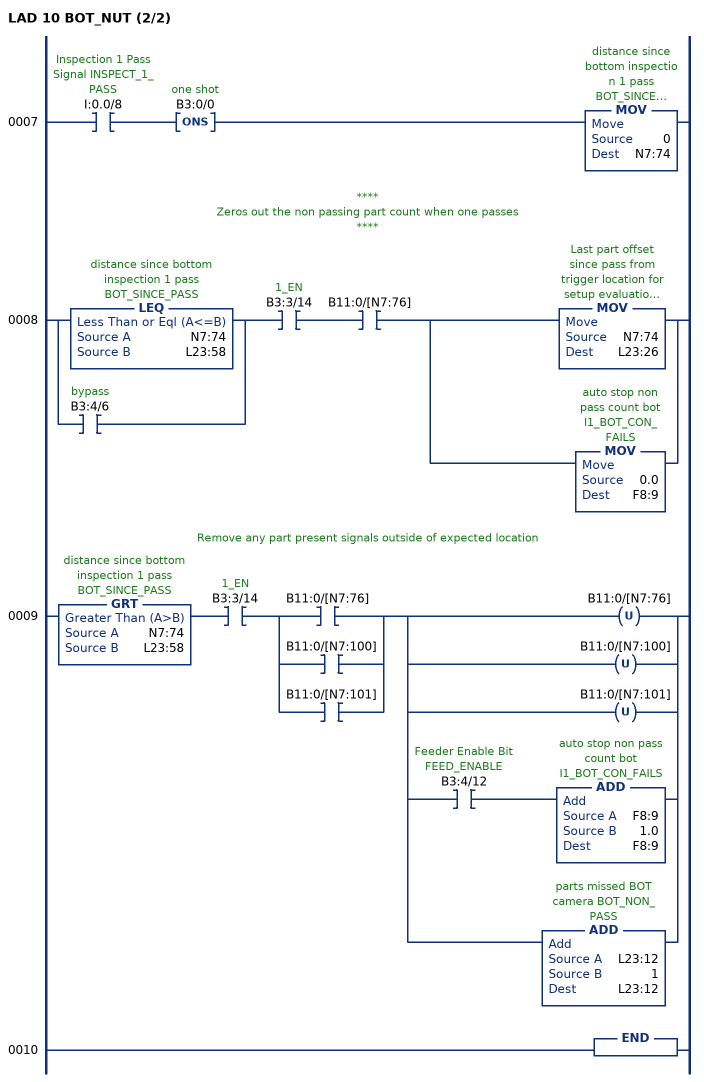
% Rung: 7 %
SOR XIC I:0.0/8 ONS B3:0/0 MOV 0 N7:74 EOR
%   I:0.0/8  INSPECT_1_PASS  "Inspection 1 Pass Signal" %
%   B3:0/0  "one shot" %
%   N7:74  BOT_SINCE_PASS  "distance since bottom inspection 1 pass" %
% Rung: 8 %
% ****
%                   Zeros out the non passing part count when one passes
% **** %
SOR BST LEQ N7:74 L23:58 NXB XIC B3:4/6 BND XIC B3:3/14 XIC B11:0/[N7:76] BST MOV N7:74 L23:26 NXB MOV 0.0 F8:9 BND EOR
%   N7:74  BOT_SINCE_PASS  "distance since bottom inspection 1 pass" %
%   L23:58  BOT_RES_WIDTH %
%   B3:4/6  "bypass" %
%   B3:3/14  1_EN %
%   N7:76  BOT_TEST_LOC  "Location of pass window." %
%   L23:26  LAST_BOT_OFFSET  "Last part offset since pass from trigger location for setup evaluation" %
%   F8:9  I1_BOT_CON_FAILS  "auto stop non pass count bot" %
% Rung: 9 %
% Remove any part present signals outside of expected location %
SOR GRT N7:74 L23:58 XIC B3:3/14 BST XIC B11:0/[N7:76] NXB XIC B11:0/[N7:100] NXB XIC B11:0/[N7:101] BND BST BST OTU B11:0/[N7:76] NXB OTU B11:0/[N7:100] NXB OTU B11:0/[N7:101] BND NXB XIC B3:4/12 ADD F8:9 1.0 F8:9 NXB ADD L23:12 1 L23:12 BND EOR
%   N7:74  BOT_SINCE_PASS  "distance since bottom inspection 1 pass" %
%   L23:58  BOT_RES_WIDTH %
%   B3:3/14  1_EN %
%   N7:76  BOT_TEST_LOC  "Location of pass window." %
%   B3:4/12  FEED_ENABLE  "Feeder Enable Bit" %
%   F8:9  I1_BOT_CON_FAILS  "auto stop non pass count bot" %
%   L23:12  BOT_NON_PASS  "parts missed BOT camera" %
% Rung: 10 %
SOR END EOR

LADDER 11 "DATA_TRANS"
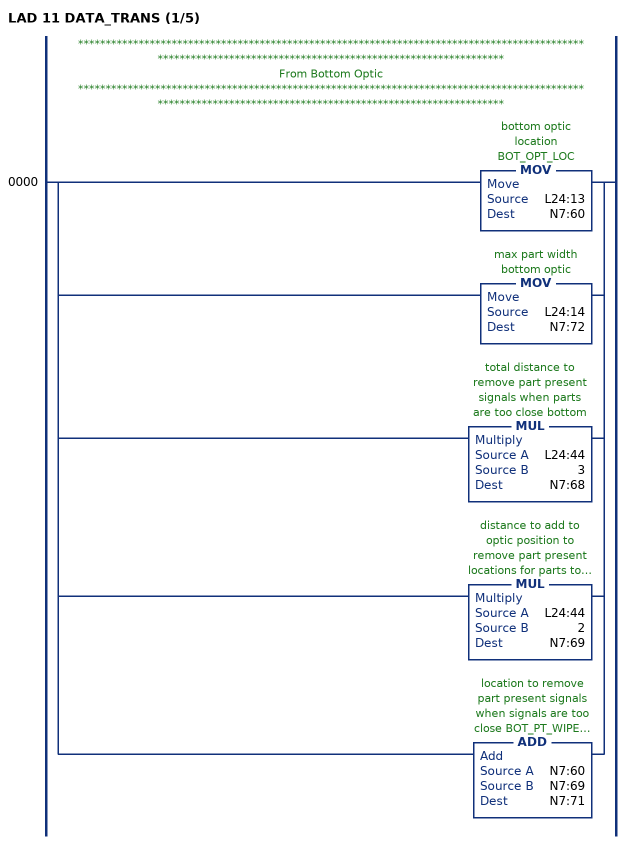
% Rung: 0 %
% ***********************************************************************************************************************************************************
% From Bottom Optic
% *********************************************************************************************************************************************************** %
SOR BST BST MOV L24:13 N7:60 NXB MOV L24:14 N7:72 BND NXB MUL L24:44 3 N7:68 NXB MUL L24:44 2 N7:69 NXB ADD N7:60 N7:69 N7:71 BND EOR
%   L24:13  BOT_OPTIC_LOC %
%   N7:60  BOT_OPT_LOC  "bottom optic location" %
%   L24:14  MAX_PART_WIDTH_BOT %
%   N7:72  "max part width bottom optic" %
%   L24:44  MIN_PART_GAP_BOT %
%   N7:68  "total distance to remove part present signals when parts are too close bottom" %
%   N7:69  "distance to add to optic position to remove part present locations for parts too close bottom" %
%   N7:71  BOT_PT_WIPE_LOC  "location to remove part present signals when signals are too close" %

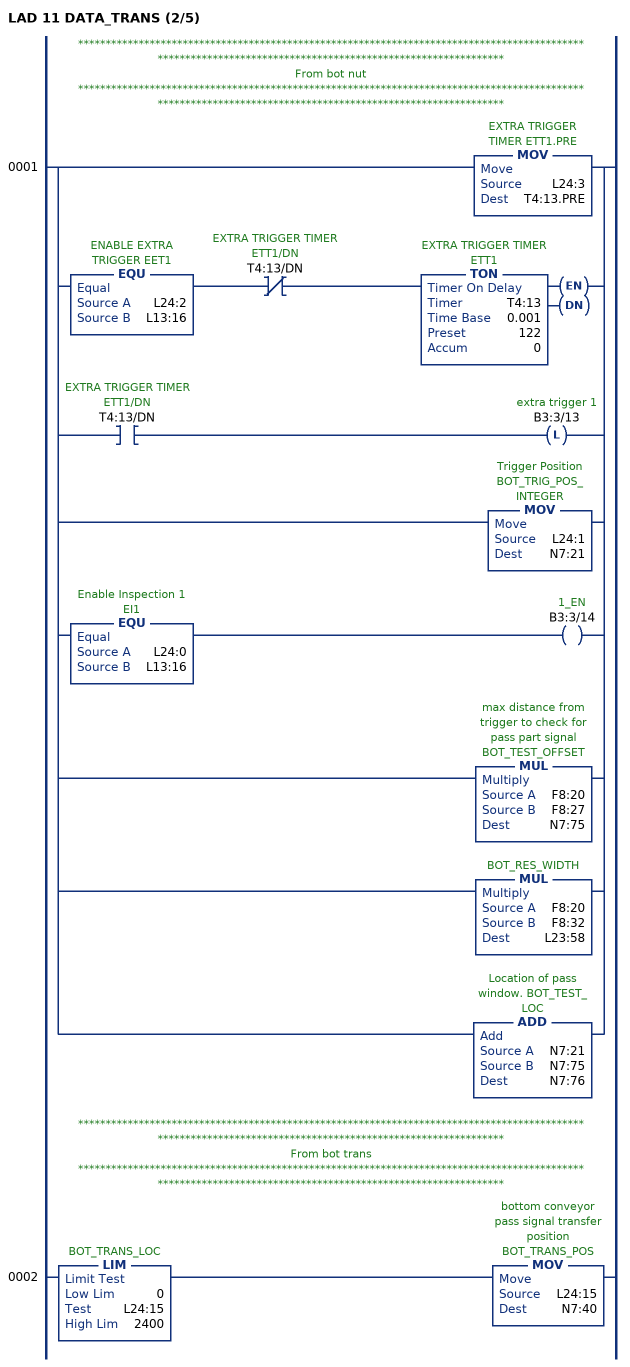
% Rung: 1 %
% ***********************************************************************************************************************************************************
% From bot nut
% *********************************************************************************************************************************************************** %
SOR BST BST MOV L24:3 T4:13.PRE NXB EQU L24:2 L13:16 XIO T4:13/DN TON T4:13 0.001 122 0 NXB XIC T4:13/DN OTL B3:3/13 NXB MOV L24:1 N7:21 NXB EQU L24:0 L13:16 OTE B3:3/14 BND NXB MUL F8:20 F8:27 N7:75 NXB MUL F8:20 F8:32 L23:58 NXB ADD N7:21 N7:75 N7:76 BND EOR
%   L24:3  ET1_DELAY %
%   T4:13  ETT1  "EXTRA TRIGGER TIMER" %
%   L24:2  EET1  "ENABLE EXTRA TRIGGER" %
%   L13:16  TRUE  "ONE TIME ENABLE FOR THE TIMES WHEN WE FORGET TO RE-ENABLE AFTER SHIPMENT" %
%   B3:3/13  "extra trigger 1" %
%   L24:1  I1_BOT_TRIG_LOC %
%   N7:21  BOT_TRIG_POS_INTEGER  "Trigger Position" %
%   L24:0  EI1  "Enable Inspection 1" %
%   B3:3/14  1_EN %
%   F8:20  "bot belt speed average in pulses per second" %
%   F8:27  MAX_TIME %
%   N7:75  BOT_TEST_OFFSET  "max distance from trigger to check for pass part signal" %
%   F8:32  TIME_WINDOW %
%   L23:58  BOT_RES_WIDTH %
%   N7:76  BOT_TEST_LOC  "Location of pass window." %
% Rung: 2 %
% ***********************************************************************************************************************************************************
% From bot trans
% *********************************************************************************************************************************************************** %
SOR LIM 0 L24:15 2400 MOV L24:15 N7:40 EOR
%   L24:15  BOT_TRANS_LOC %
%   N7:40  BOT_TRANS_POS  "bottom conveyor pass signal transfer position" %

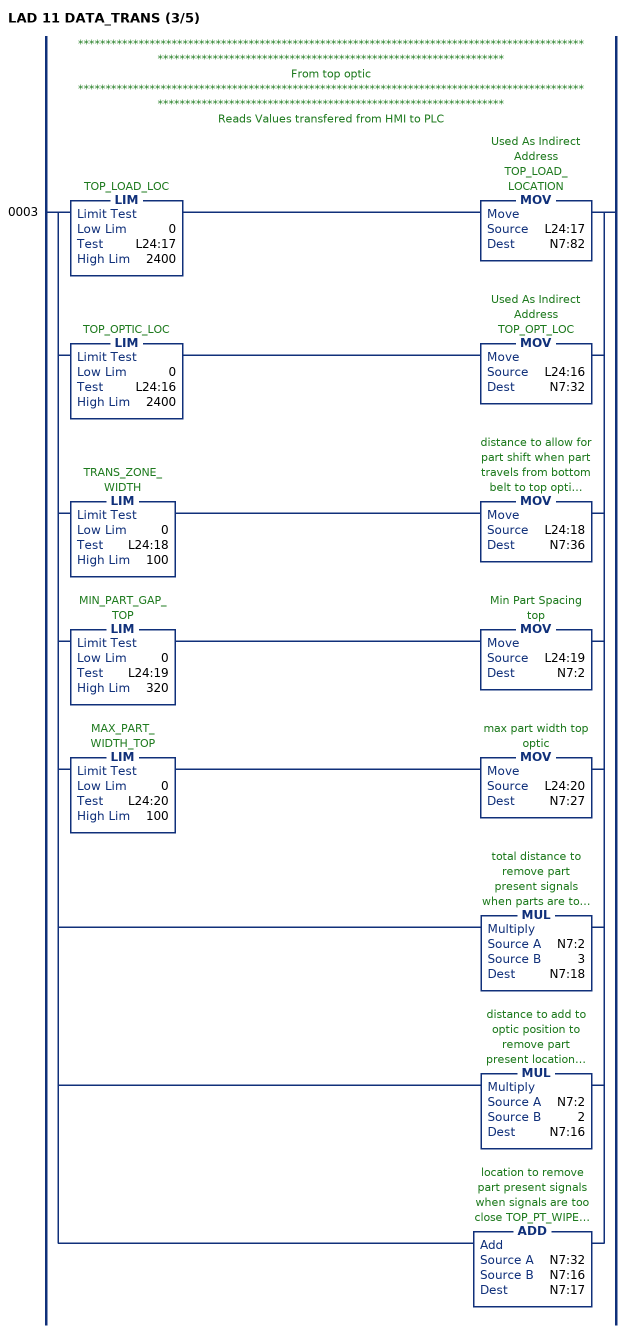
% Rung: 3 %
% ***********************************************************************************************************************************************************
% From top optic
% ***********************************************************************************************************************************************************
% 
% Reads Values transfered from HMI to PLC %
SOR BST BST LIM 0 L24:17 2400 MOV L24:17 N7:82 NXB LIM 0 L24:16 2400 MOV L24:16 N7:32 NXB LIM 0 L24:18 100 MOV L24:18 N7:36 NXB LIM 0 L24:19 320 MOV L24:19 N7:2 NXB LIM 0 L24:20 100 MOV L24:20 N7:27 BND NXB MUL N7:2 3 N7:18 NXB MUL N7:2 2 N7:16 NXB ADD N7:32 N7:16 N7:17 BND EOR
%   L24:17  TOP_LOAD_LOC %
%   N7:82  TOP_LOAD_LOCATION  "Used As Indirect Address" %
%   L24:16  TOP_OPTIC_LOC %
%   N7:32  TOP_OPT_LOC  "Used As Indirect Address" %
%   L24:18  TRANS_ZONE_WIDTH %
%   N7:36  TRANS_ZONE  "distance to allow for part shift when part travels from bottom belt to top optic" %
%   L24:19  MIN_PART_GAP_TOP %
%   N7:2  "Min Part Spacing top" %
%   L24:20  MAX_PART_WIDTH_TOP %
%   N7:27  "max part width top optic" %
%   N7:18  "total distance to remove part present signals when parts are too close top" %
%   N7:16  "distance to add to optic position to remove part present locations for parts too close top" %
%   N7:17  TOP_PT_WIPE_LOC  "location to remove part present signals when signals are too close" %

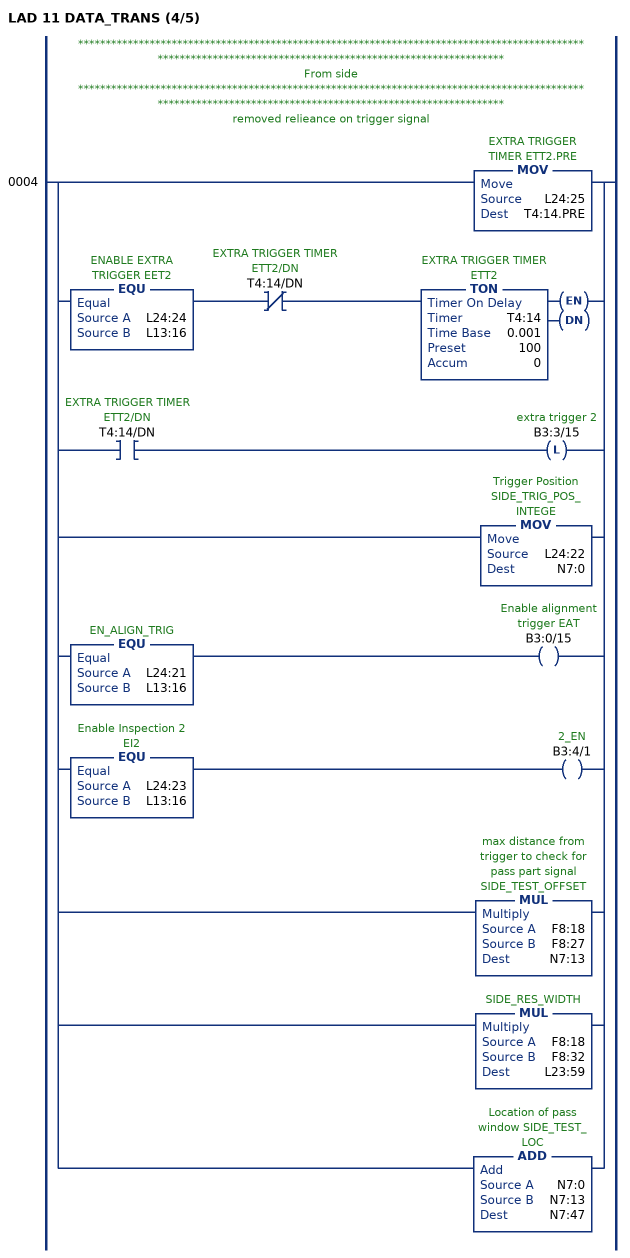
% Rung: 4 %
% ***********************************************************************************************************************************************************
% From side
% ***********************************************************************************************************************************************************
% 
% removed relieance on trigger signal %
SOR BST BST MOV L24:25 T4:14.PRE NXB EQU L24:24 L13:16 XIO T4:14/DN TON T4:14 0.001 100 0 NXB XIC T4:14/DN OTL B3:3/15 NXB MOV L24:22 N7:0 NXB EQU L24:21 L13:16 OTE B3:0/15 NXB EQU L24:23 L13:16 OTE B3:4/1 BND NXB MUL F8:18 F8:27 N7:13 NXB MUL F8:18 F8:32 L23:59 NXB ADD N7:0 N7:13 N7:47 BND EOR
%   L24:25  ET2_DELAY %
%   T4:14  ETT2  "EXTRA TRIGGER TIMER" %
%   L24:24  EET2  "ENABLE EXTRA TRIGGER" %
%   L13:16  TRUE  "ONE TIME ENABLE FOR THE TIMES WHEN WE FORGET TO RE-ENABLE AFTER SHIPMENT" %
%   B3:3/15  "extra trigger 2" %
%   L24:22  I2_SIDE_TRIG_LOC %
%   N7:0  SIDE_TRIG_POS_INTEGE  "Trigger Position" %
%   L24:21  EN_ALIGN_TRIG %
%   B3:0/15  EAT  "Enable alignment trigger" %
%   L24:23  EI2  "Enable Inspection 2" %
%   B3:4/1  2_EN %
%   F8:18  "top belt speed average in pulses per second 290 Max; Verify" %
%   F8:27  MAX_TIME %
%   N7:13  SIDE_TEST_OFFSET  "max distance from trigger to check for pass part signal" %
%   F8:32  TIME_WINDOW %
%   L23:59  SIDE_RES_WIDTH %
%   N7:47  SIDE_TEST_LOC  "Location of pass window" %

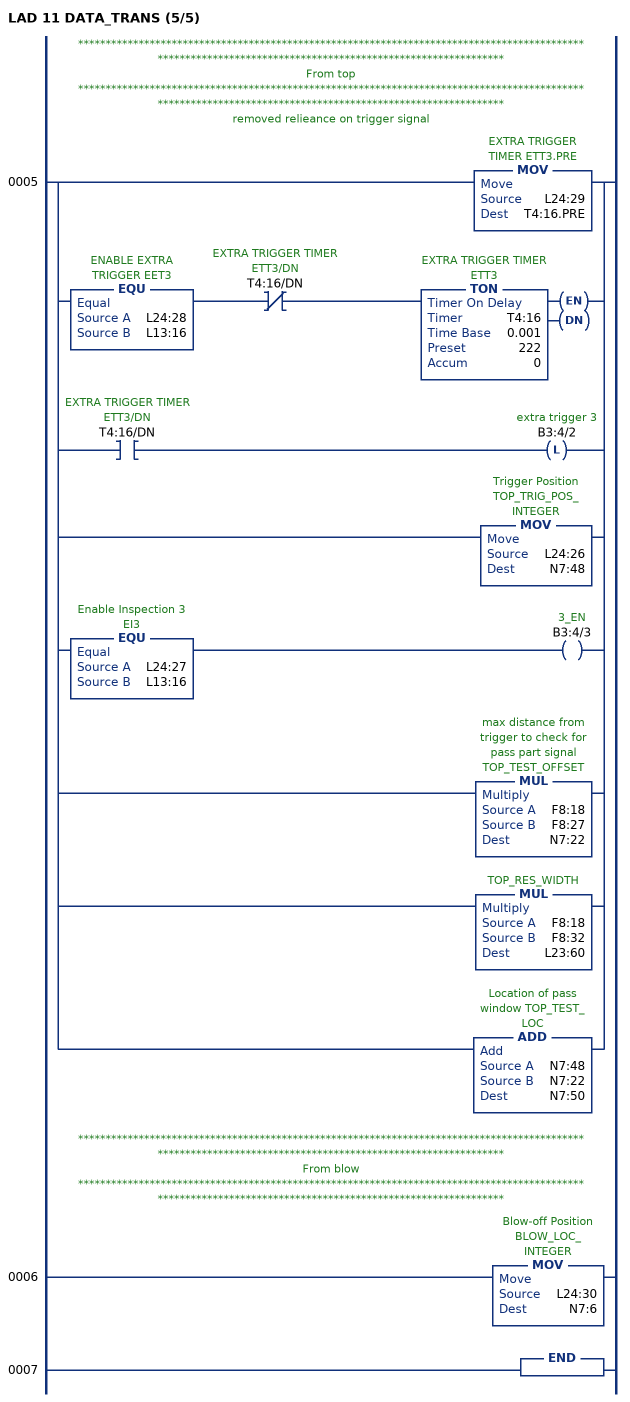
% Rung: 5 %
% ***********************************************************************************************************************************************************
% From top
% ***********************************************************************************************************************************************************
% 
% removed relieance on trigger signal %
SOR BST BST MOV L24:29 T4:16.PRE NXB EQU L24:28 L13:16 XIO T4:16/DN TON T4:16 0.001 222 0 NXB XIC T4:16/DN OTL B3:4/2 NXB MOV L24:26 N7:48 NXB EQU L24:27 L13:16 OTE B3:4/3 BND NXB MUL F8:18 F8:27 N7:22 NXB MUL F8:18 F8:32 L23:60 NXB ADD N7:48 N7:22 N7:50 BND EOR
%   L24:29  ET3_DELAY %
%   T4:16  ETT3  "EXTRA TRIGGER TIMER" %
%   L24:28  EET3  "ENABLE EXTRA TRIGGER" %
%   L13:16  TRUE  "ONE TIME ENABLE FOR THE TIMES WHEN WE FORGET TO RE-ENABLE AFTER SHIPMENT" %
%   B3:4/2  "extra trigger 3" %
%   L24:26  I3_TOP_TRIG_LOC %
%   N7:48  TOP_TRIG_POS_INTEGER  "Trigger Position" %
%   L24:27  EI3  "Enable Inspection 3" %
%   B3:4/3  3_EN %
%   F8:18  "top belt speed average in pulses per second 290 Max; Verify" %
%   F8:27  MAX_TIME %
%   N7:22  TOP_TEST_OFFSET  "max distance from trigger to check for pass part signal" %
%   F8:32  TIME_WINDOW %
%   L23:60  TOP_RES_WIDTH %
%   N7:50  TOP_TEST_LOC  "Location of pass window" %
% Rung: 6 %
% ***********************************************************************************************************************************************************
% From blow
% *********************************************************************************************************************************************************** %
SOR MOV L24:30 N7:6 EOR
%   L24:30  BLOW_OFF_LOC %
%   N7:6  BLOW_LOC_INTEGER  "Blow-off Position" %
% Rung: 7 %
SOR END EOR

LADDER 12 "BOT_TRANSF"
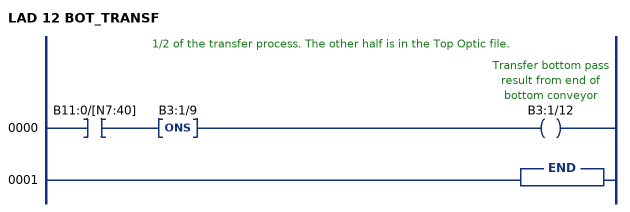
% Rung: 0 %
% 1/2 of the transfer process. The other half is in the Top Optic file. %
SOR XIC B11:0/[N7:40] ONS B3:1/9 OTE B3:1/12 EOR
%   N7:40  BOT_TRANS_POS  "bottom conveyor pass signal transfer position" %
%   B3:1/12  "Transfer bottom pass result from end of bottom conveyor" %
% Rung: 1 %
SOR END EOR

LADDER 14 "TOP_OPTIC"
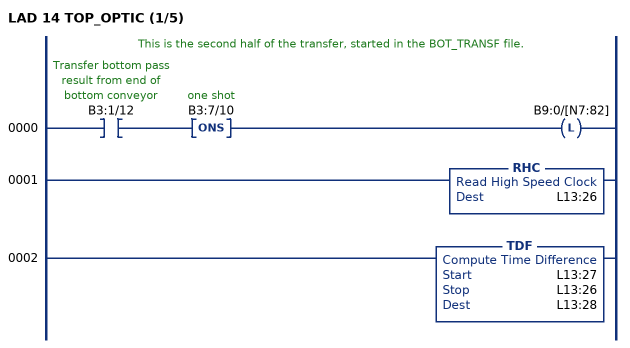
% Rung: 0 %
% This is the second half of the transfer, started in the BOT_TRANSF file. %
SOR XIC B3:1/12 ONS B3:7/10 OTL B9:0/[N7:82] EOR
%   B3:1/12  "Transfer bottom pass result from end of bottom conveyor" %
%   B3:7/10  "one shot" %
%   N7:82  TOP_LOAD_LOCATION  "Used As Indirect Address" %
% Rung: 1 %
SOR RHC L13:26 EOR
% Rung: 2 %
SOR TDF L13:27 L13:26 L13:28 EOR

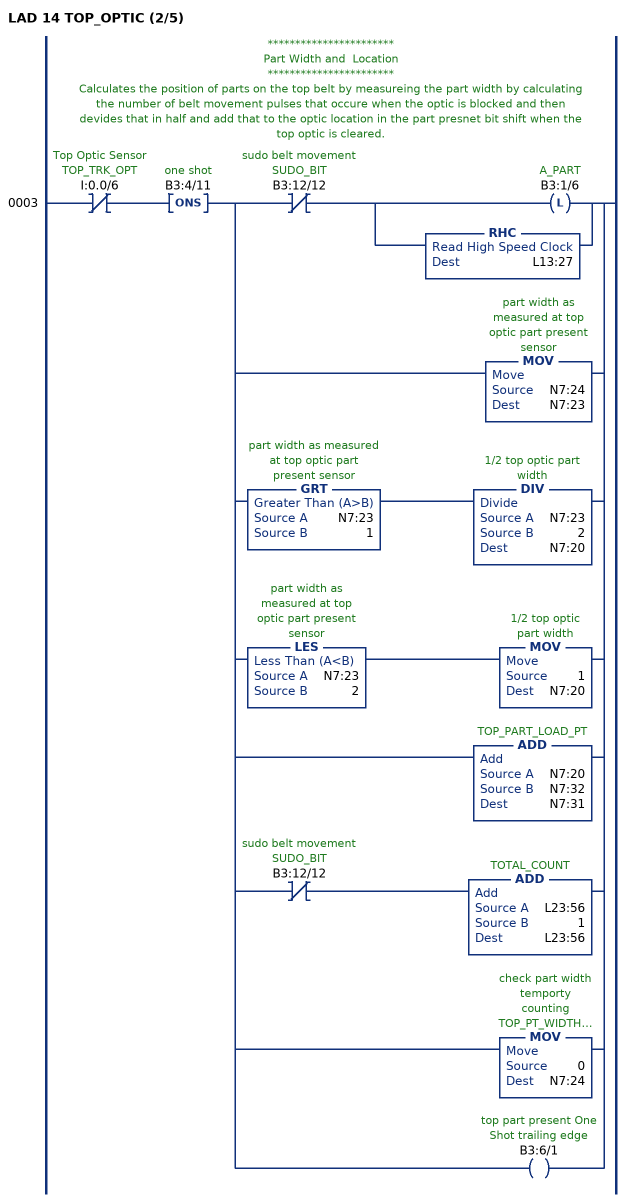
% Rung: 3 %
% ***********************
% Part Width and  Location
% ***********************
% 
% Calculates the position of parts on the top belt by measureing the part width by calculating the number of belt movement pulses that occure when the optic is blocked and then devides that in half and add that to the optic location in the part presnet bit shift when the top optic is cleared. %
SOR XIO I:0.0/6 ONS B3:4/11 BST XIO B3:12/12 BST OTL B3:1/6 NXB RHC L13:27 BND NXB MOV N7:24 N7:23 NXB GRT N7:23 1 DIV N7:23 2 N7:20 NXB LES N7:23 2 MOV 1 N7:20 NXB ADD N7:20 N7:32 N7:31 NXB XIO B3:12/12 ADD L23:56 1 L23:56 NXB MOV 0 N7:24 NXB OTE B3:6/1 BND EOR
%   I:0.0/6  TOP_TRK_OPT  "Top Optic Sensor" %
%   B3:4/11  "one shot" %
%   B3:12/12  SUDO_BIT  "sudo belt movement" %
%   B3:1/6  A_PART %
%   N7:24  TOP_PT_WIDTH_TEMP  "check part width temporty counting" %
%   N7:23  "part width as measured at top optic part present sensor" %
%   N7:20  "1/2 top optic part width" %
%   N7:32  TOP_OPT_LOC  "Used As Indirect Address" %
%   N7:31  TOP_PART_LOAD_PT %
%   L23:56  TOTAL_COUNT %
%   B3:6/1  "top part present One Shot trailing edge" %

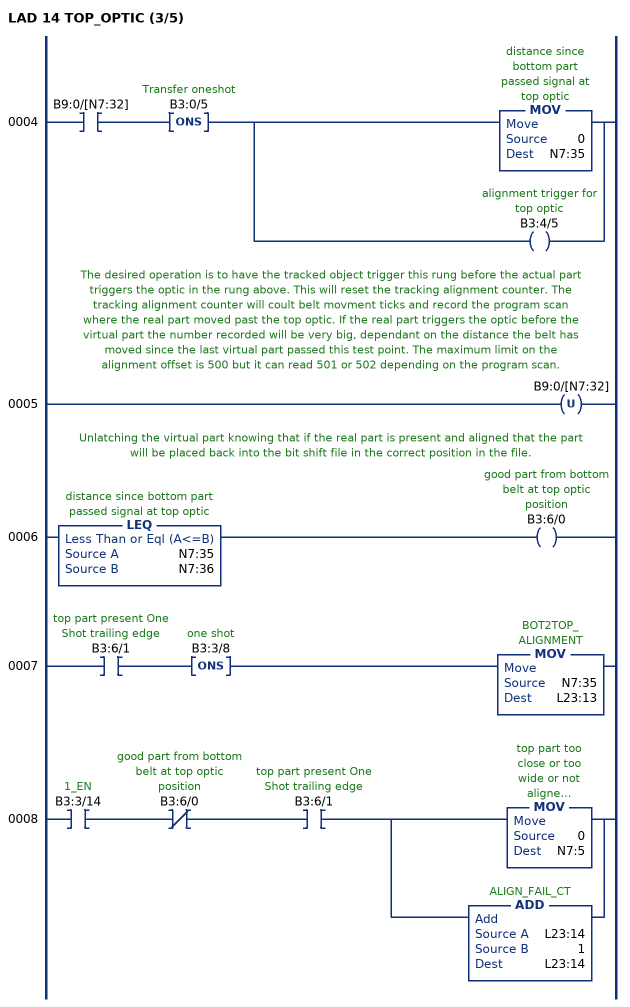
% Rung: 4 %
SOR XIC B9:0/[N7:32] ONS B3:0/5 BST MOV 0 N7:35 NXB OTE B3:4/5 BND EOR
%   N7:32  TOP_OPT_LOC  "Used As Indirect Address" %
%   B3:0/5  "Transfer oneshot" %
%   N7:35  "distance since bottom part passed signal at top optic" %
%   B3:4/5  "alignment trigger for top optic" %
% Rung: 5 %
% The desired operation is to have the tracked object trigger this rung before the actual part triggers the optic in the rung above. This will reset the tracking alignment counter. The tracking alignment counter will coult belt movment ticks and record the program scan where the real part moved past the top optic. If the real part triggers the optic before the virtual part the number recorded will be very big, dependant on the distance the belt has moved since the last virtual part passed this test point. The maximum limit on the alignment offset is 500 but it can read 501 or 502 depending on the program scan. %
SOR OTU B9:0/[N7:32] EOR
%   N7:32  TOP_OPT_LOC  "Used As Indirect Address" %
% Rung: 6 %
% Unlatching the virtual part knowing that if the real part is present and aligned that the part will be placed back into the bit shift file in the correct position in the file. %
SOR LEQ N7:35 N7:36 OTE B3:6/0 EOR
%   N7:35  "distance since bottom part passed signal at top optic" %
%   N7:36  TRANS_ZONE  "distance to allow for part shift when part travels from bottom belt to top optic" %
%   B3:6/0  "good part from bottom belt at top optic position" %
% Rung: 7 %
SOR XIC B3:6/1 ONS B3:3/8 MOV N7:35 L23:13 EOR
%   B3:6/1  "top part present One Shot trailing edge" %
%   B3:3/8  "one shot" %
%   N7:35  "distance since bottom part passed signal at top optic" %
%   L23:13  BOT2TOP_ALIGNMENT %
% Rung: 8 %
SOR XIC B3:3/14 XIO B3:6/0 XIC B3:6/1 BST MOV 0 N7:5 NXB ADD L23:14 1 L23:14 BND EOR
%   B3:3/14  1_EN %
%   B3:6/0  "good part from bottom belt at top optic position" %
%   B3:6/1  "top part present One Shot trailing edge" %
%   N7:5  "top part too close or too wide or not aligned distance measurement" %
%   L23:14  ALIGN_FAIL_CT %

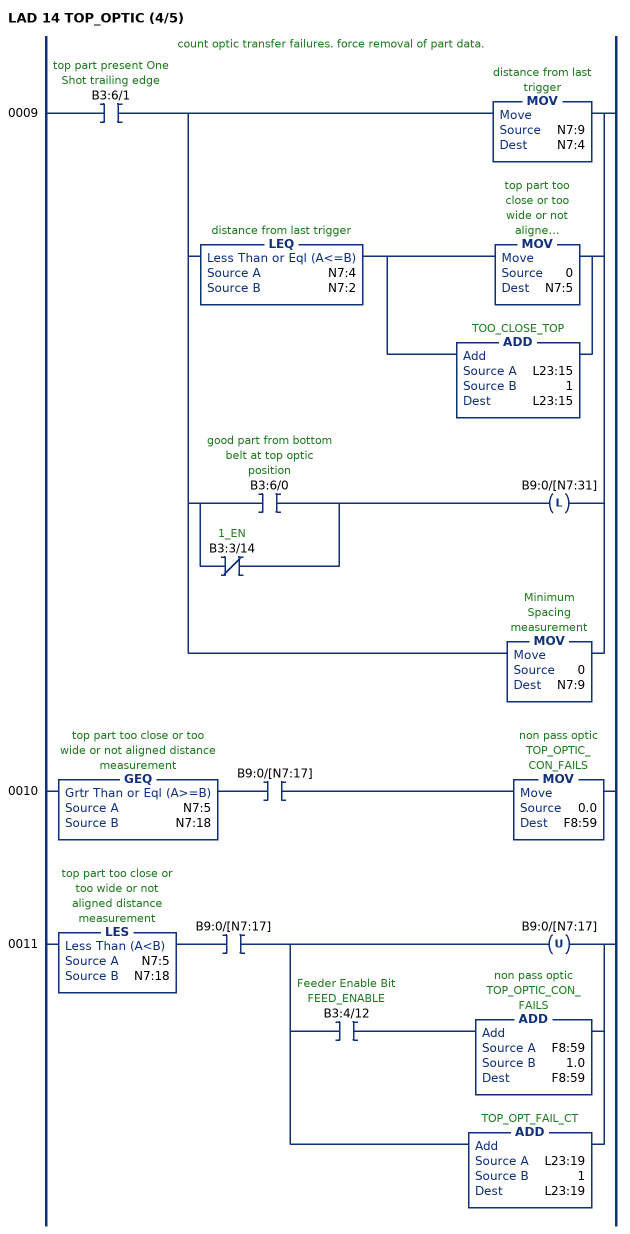
% Rung: 9 %
% count optic transfer failures. force removal of part data. %
SOR XIC B3:6/1 BST MOV N7:9 N7:4 NXB LEQ N7:4 N7:2 BST MOV 0 N7:5 NXB ADD L23:15 1 L23:15 BND NXB BST XIC B3:6/0 NXB XIO B3:3/14 BND OTL B9:0/[N7:31] NXB MOV 0 N7:9 BND EOR
%   B3:6/1  "top part present One Shot trailing edge" %
%   N7:9  "Minimum Spacing measurement" %
%   N7:4  "distance from last trigger" %
%   N7:2  "Min Part Spacing top" %
%   N7:5  "top part too close or too wide or not aligned distance measurement" %
%   L23:15  TOO_CLOSE_TOP %
%   B3:6/0  "good part from bottom belt at top optic position" %
%   B3:3/14  1_EN %
%   N7:31  TOP_PART_LOAD_PT %
% Rung: 10 %
SOR GEQ N7:5 N7:18 XIC B9:0/[N7:17] MOV 0.0 F8:59 EOR
%   N7:5  "top part too close or too wide or not aligned distance measurement" %
%   N7:18  "total distance to remove part present signals when parts are too close top" %
%   N7:17  TOP_PT_WIPE_LOC  "location to remove part present signals when signals are too close" %
%   F8:59  TOP_OPTIC_CON_FAILS  "non pass optic" %
% Rung: 11 %
SOR LES N7:5 N7:18 XIC B9:0/[N7:17] BST OTU B9:0/[N7:17] NXB XIC B3:4/12 ADD F8:59 1.0 F8:59 NXB ADD L23:19 1 L23:19 BND EOR
%   N7:5  "top part too close or too wide or not aligned distance measurement" %
%   N7:18  "total distance to remove part present signals when parts are too close top" %
%   N7:17  TOP_PT_WIPE_LOC  "location to remove part present signals when signals are too close" %
%   B3:4/12  FEED_ENABLE  "Feeder Enable Bit" %
%   F8:59  TOP_OPTIC_CON_FAILS  "non pass optic" %
%   L23:19  TOP_OPT_FAIL_CT %

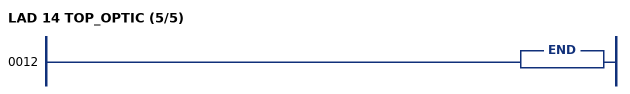
% Rung: 12 %
SOR END EOR

LADDER 16 "TOP_SIDE"
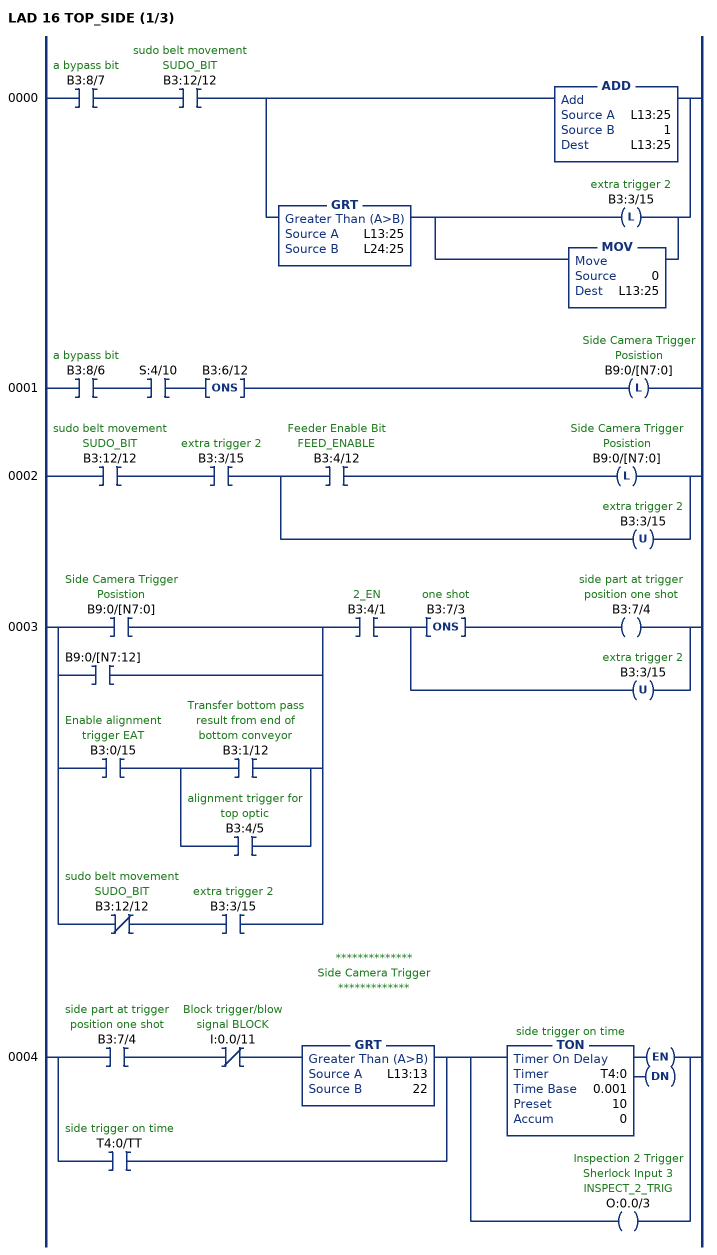
% Rung: 0 %
SOR XIC B3:8/7 XIC B3:12/12 BST ADD L13:25 1 L13:25 NXB GRT L13:25 L24:25 BST OTL B3:3/15 NXB MOV 0 L13:25 BND BND EOR
%   B3:8/7  "a bypass bit" %
%   B3:12/12  SUDO_BIT  "sudo belt movement" %
%   L24:25  ET2_DELAY %
%   B3:3/15  "extra trigger 2" %
% Rung: 1 %
SOR XIC B3:8/6 XIC S:4/10 ONS B3:6/12 OTL B9:0/[N7:0] EOR
%   B3:8/6  "a bypass bit" %
%   B9:0/[N7:0]  "Side Camera Trigger Posistion" %
%   N7:0  SIDE_TRIG_POS_INTEGE  "Trigger Position" %
% Rung: 2 %
SOR XIC B3:12/12 XIC B3:3/15 BST XIC B3:4/12 OTL B9:0/[N7:0] NXB OTU B3:3/15 BND EOR
%   B3:12/12  SUDO_BIT  "sudo belt movement" %
%   B3:3/15  "extra trigger 2" %
%   B3:4/12  FEED_ENABLE  "Feeder Enable Bit" %
%   B9:0/[N7:0]  "Side Camera Trigger Posistion" %
%   N7:0  SIDE_TRIG_POS_INTEGE  "Trigger Position" %
% Rung: 3 %
SOR BST XIC B9:0/[N7:0] NXB XIC B9:0/[N7:12] NXB XIC B3:0/15 BST XIC B3:1/12 NXB XIC B3:4/5 BND NXB XIO B3:12/12 XIC B3:3/15 BND XIC B3:4/1 BST ONS B3:7/3 OTE B3:7/4 NXB OTU B3:3/15 BND EOR
%   B9:0/[N7:0]  "Side Camera Trigger Posistion" %
%   N7:0  SIDE_TRIG_POS_INTEGE  "Trigger Position" %
%   N7:12  "second side trigger position" %
%   B3:0/15  EAT  "Enable alignment trigger" %
%   B3:1/12  "Transfer bottom pass result from end of bottom conveyor" %
%   B3:4/5  "alignment trigger for top optic" %
%   B3:12/12  SUDO_BIT  "sudo belt movement" %
%   B3:3/15  "extra trigger 2" %
%   B3:4/1  2_EN %
%   B3:7/3  "one shot" %
%   B3:7/4  "side part at trigger position one shot" %
% Rung: 4 %
% **************
% Side Camera Trigger
% ************* %
SOR BST XIC B3:7/4 XIO I:0.0/11 GRT L13:13 22 NXB XIC T4:0/TT BND BST TON T4:0 0.001 10 0 NXB OTE O:0.0/3 BND EOR
%   B3:7/4  "side part at trigger position one shot" %
%   I:0.0/11  BLOCK  "Block trigger/blow signal" %
%   T4:0  "side trigger on time" %
%   O:0.0/3  INSPECT_2_TRIG  "Inspection 2 Trigger Sherlock Input 3" %

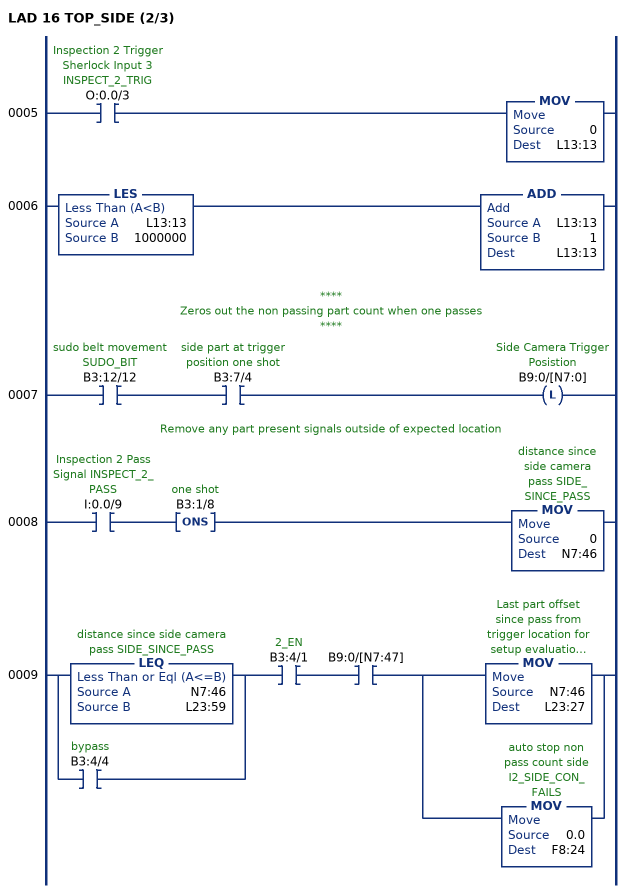
% Rung: 5 %
SOR XIC O:0.0/3 MOV 0 L13:13 EOR
%   O:0.0/3  INSPECT_2_TRIG  "Inspection 2 Trigger Sherlock Input 3" %
% Rung: 6 %
SOR LES L13:13 1000000 ADD L13:13 1 L13:13 EOR
% Rung: 7 %
% ****
%                   Zeros out the non passing part count when one passes
% **** %
SOR XIC B3:12/12 XIC B3:7/4 OTL B9:0/[N7:0] EOR
%   B3:12/12  SUDO_BIT  "sudo belt movement" %
%   B3:7/4  "side part at trigger position one shot" %
%   B9:0/[N7:0]  "Side Camera Trigger Posistion" %
%   N7:0  SIDE_TRIG_POS_INTEGE  "Trigger Position" %
% Rung: 8 %
% Remove any part present signals outside of expected location %
SOR XIC I:0.0/9 ONS B3:1/8 MOV 0 N7:46 EOR
%   I:0.0/9  INSPECT_2_PASS  "Inspection 2 Pass Signal" %
%   B3:1/8  "one shot" %
%   N7:46  SIDE_SINCE_PASS  "distance since side camera pass" %
% Rung: 9 %
SOR BST LEQ N7:46 L23:59 NXB XIC B3:4/4 BND XIC B3:4/1 XIC B9:0/[N7:47] BST MOV N7:46 L23:27 NXB MOV 0.0 F8:24 BND EOR
%   N7:46  SIDE_SINCE_PASS  "distance since side camera pass" %
%   L23:59  SIDE_RES_WIDTH %
%   B3:4/4  "bypass" %
%   B3:4/1  2_EN %
%   N7:47  SIDE_TEST_LOC  "Location of pass window" %
%   L23:27  LAST_SIDE_OFFSET  "Last part offset since pass from trigger location for setup evaluation" %
%   F8:24  I2_SIDE_CON_FAILS  "auto stop non pass count side" %

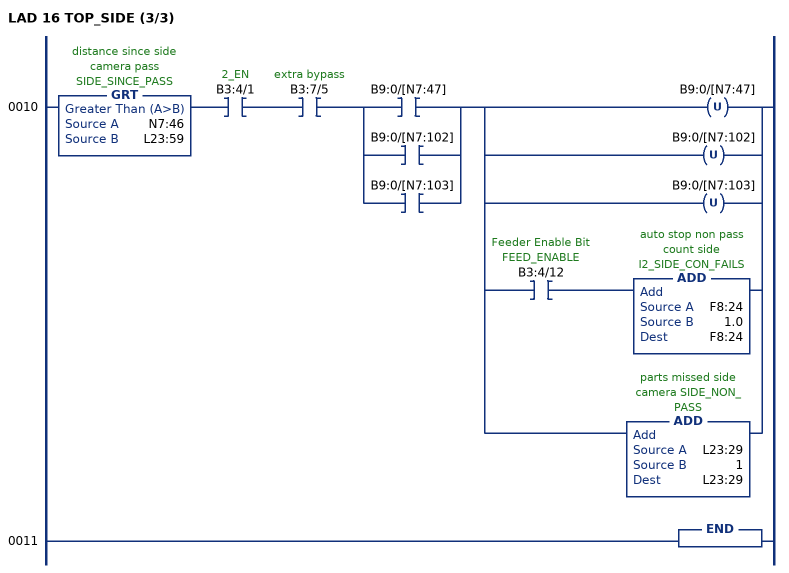
% Rung: 10 %
SOR GRT N7:46 L23:59 XIC B3:4/1 XIC B3:7/5 BST XIC B9:0/[N7:47] NXB XIC B9:0/[N7:102] NXB XIC B9:0/[N7:103] BND BST BST OTU B9:0/[N7:47] NXB OTU B9:0/[N7:102] NXB OTU B9:0/[N7:103] BND NXB XIC B3:4/12 ADD F8:24 1.0 F8:24 NXB ADD L23:29 1 L23:29 BND EOR
%   N7:46  SIDE_SINCE_PASS  "distance since side camera pass" %
%   L23:59  SIDE_RES_WIDTH %
%   B3:4/1  2_EN %
%   B3:7/5  "extra bypass" %
%   N7:47  SIDE_TEST_LOC  "Location of pass window" %
%   B3:4/12  FEED_ENABLE  "Feeder Enable Bit" %
%   F8:24  I2_SIDE_CON_FAILS  "auto stop non pass count side" %
%   L23:29  SIDE_NON_PASS  "parts missed side camera" %
% Rung: 11 %
SOR END EOR

LADDER 20 "TOP_TOP"
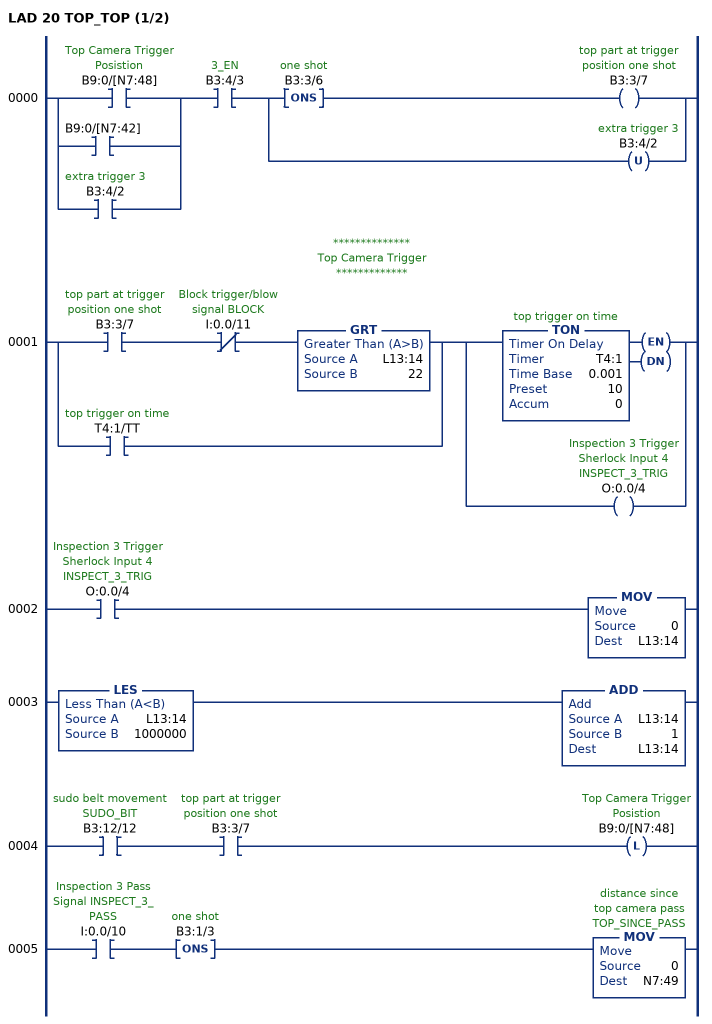
% Rung: 0 %
SOR BST XIC B9:0/[N7:48] NXB XIC B9:0/[N7:42] NXB XIC B3:4/2 BND XIC B3:4/3 BST ONS B3:3/6 OTE B3:3/7 NXB OTU B3:4/2 BND EOR
%   B9:0/[N7:48]  "Top Camera Trigger Posistion" %
%   N7:48  TOP_TRIG_POS_INTEGER  "Trigger Position" %
%   N7:42  "second top trigger position" %
%   B3:4/2  "extra trigger 3" %
%   B3:4/3  3_EN %
%   B3:3/6  "one shot" %
%   B3:3/7  "top part at trigger position one shot" %
% Rung: 1 %
% **************
% Top Camera Trigger
% ************* %
SOR BST XIC B3:3/7 XIO I:0.0/11 GRT L13:14 22 NXB XIC T4:1/TT BND BST TON T4:1 0.001 10 0 NXB OTE O:0.0/4 BND EOR
%   B3:3/7  "top part at trigger position one shot" %
%   I:0.0/11  BLOCK  "Block trigger/blow signal" %
%   T4:1  "top trigger on time" %
%   O:0.0/4  INSPECT_3_TRIG  "Inspection 3 Trigger Sherlock Input 4" %
% Rung: 2 %
SOR XIC O:0.0/4 MOV 0 L13:14 EOR
%   O:0.0/4  INSPECT_3_TRIG  "Inspection 3 Trigger Sherlock Input 4" %
% Rung: 3 %
SOR LES L13:14 1000000 ADD L13:14 1 L13:14 EOR
% Rung: 4 %
SOR XIC B3:12/12 XIC B3:3/7 OTL B9:0/[N7:48] EOR
%   B3:12/12  SUDO_BIT  "sudo belt movement" %
%   B3:3/7  "top part at trigger position one shot" %
%   B9:0/[N7:48]  "Top Camera Trigger Posistion" %
%   N7:48  TOP_TRIG_POS_INTEGER  "Trigger Position" %
% Rung: 5 %
SOR XIC I:0.0/10 ONS B3:1/3 MOV 0 N7:49 EOR
%   I:0.0/10  INSPECT_3_PASS  "Inspection 3 Pass Signal" %
%   B3:1/3  "one shot" %
%   N7:49  TOP_SINCE_PASS  "distance since top camera pass" %

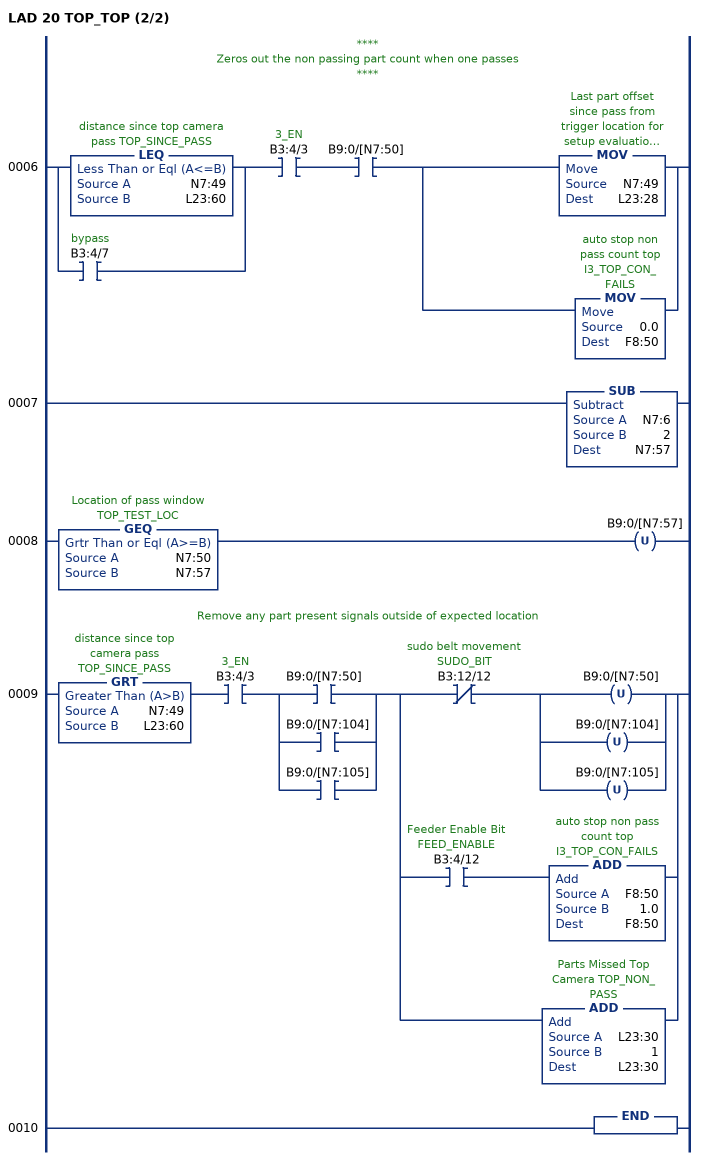
% Rung: 6 %
% ****
%                   Zeros out the non passing part count when one passes
% **** %
SOR BST LEQ N7:49 L23:60 NXB XIC B3:4/7 BND XIC B3:4/3 XIC B9:0/[N7:50] BST MOV N7:49 L23:28 NXB MOV 0.0 F8:50 BND EOR
%   N7:49  TOP_SINCE_PASS  "distance since top camera pass" %
%   L23:60  TOP_RES_WIDTH %
%   B3:4/7  "bypass" %
%   B3:4/3  3_EN %
%   N7:50  TOP_TEST_LOC  "Location of pass window" %
%   L23:28  LAST_TOP_OFFSET  "Last part offset since pass from trigger location for setup evaluation" %
%   F8:50  I3_TOP_CON_FAILS  "auto stop non pass count top" %
% Rung: 7 %
SOR SUB N7:6 2 N7:57 EOR
%   N7:6  BLOW_LOC_INTEGER  "Blow-off Position" %
% Rung: 8 %
SOR GEQ N7:50 N7:57 OTU B9:0/[N7:57] EOR
%   N7:50  TOP_TEST_LOC  "Location of pass window" %
% Rung: 9 %
% Remove any part present signals outside of expected location %
SOR GRT N7:49 L23:60 XIC B3:4/3 BST XIC B9:0/[N7:50] NXB XIC B9:0/[N7:104] NXB XIC B9:0/[N7:105] BND BST XIO B3:12/12 BST OTU B9:0/[N7:50] NXB OTU B9:0/[N7:104] NXB OTU B9:0/[N7:105] BND NXB XIC B3:4/12 ADD F8:50 1.0 F8:50 NXB ADD L23:30 1 L23:30 BND EOR
%   N7:49  TOP_SINCE_PASS  "distance since top camera pass" %
%   L23:60  TOP_RES_WIDTH %
%   B3:4/3  3_EN %
%   N7:50  TOP_TEST_LOC  "Location of pass window" %
%   B3:12/12  SUDO_BIT  "sudo belt movement" %
%   B3:4/12  FEED_ENABLE  "Feeder Enable Bit" %
%   F8:50  I3_TOP_CON_FAILS  "auto stop non pass count top" %
%   L23:30  TOP_NON_PASS  "Parts Missed Top Camera" %
% Rung: 10 %
SOR END EOR

LADDER 24 "TOP_BLOW"
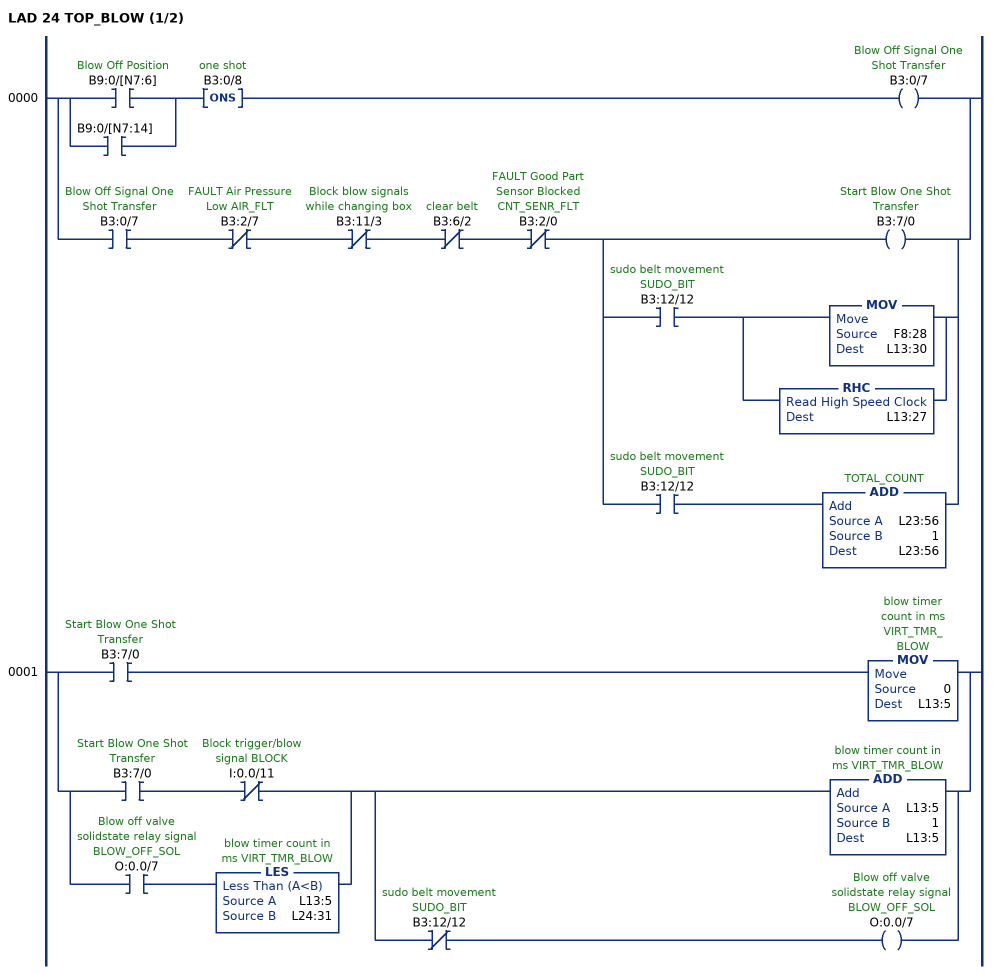
% Rung: 0 %
SOR BST BST XIC B9:0/[N7:6] NXB XIC B9:0/[N7:14] BND ONS B3:0/8 OTE B3:0/7 NXB XIC B3:0/7 XIO B3:2/7 XIO B3:11/3 XIO B3:6/2 XIO B3:2/0 BST OTE B3:7/0 NXB XIC B3:12/12 BST MOV F8:28 L13:30 NXB RHC L13:27 BND NXB XIC B3:12/12 ADD L23:56 1 L23:56 BND BND EOR
%   B9:0/[N7:6]  "Blow Off Position" %
%   N7:6  BLOW_LOC_INTEGER  "Blow-off Position" %
%   N7:14  "second blow position" %
%   B3:0/8  "one shot" %
%   B3:0/7  "Blow Off Signal One Shot Transfer" %
%   B3:2/7  AIR_FLT  "FAULT Air Pressure Low" %
%   B3:11/3  "Block blow signals while changing box" %
%   B3:6/2  "clear belt" %
%   B3:2/0  CNT_SENR_FLT  "FAULT Good Part Sensor Blocked" %
%   B3:7/0  "Start Blow One Shot Transfer" %
%   B3:12/12  SUDO_BIT  "sudo belt movement" %
%   F8:28  "momentary rate in ppm" %
%   L23:56  TOTAL_COUNT %
% Rung: 1 %
SOR BST XIC B3:7/0 MOV 0 L13:5 NXB BST XIC B3:7/0 XIO I:0.0/11 NXB XIC O:0.0/7 LES L13:5 L24:31 BND BST ADD L13:5 1 L13:5 NXB XIO B3:12/12 OTE O:0.0/7 BND BND EOR
%   B3:7/0  "Start Blow One Shot Transfer" %
%   L13:5  VIRT_TMR_BLOW  "blow timer count in ms" %
%   I:0.0/11  BLOCK  "Block trigger/blow signal" %
%   O:0.0/7  BLOW_OFF_SOL  "Blow off valve solidstate relay signal" %
%   L24:31  BLOW_TIME %
%   B3:12/12  SUDO_BIT  "sudo belt movement" %

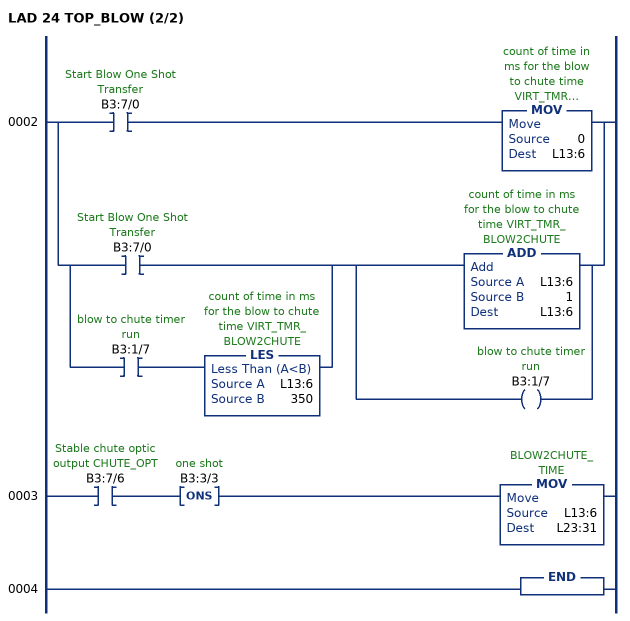
% Rung: 2 %
SOR BST XIC B3:7/0 MOV 0 L13:6 NXB BST XIC B3:7/0 NXB XIC B3:1/7 LES L13:6 350 BND BST ADD L13:6 1 L13:6 NXB OTE B3:1/7 BND BND EOR
%   B3:7/0  "Start Blow One Shot Transfer" %
%   L13:6  VIRT_TMR_BLOW2CHUTE  "count of time in ms for the blow to chute time" %
%   B3:1/7  "blow to chute timer run" %
% Rung: 3 %
SOR XIC B3:7/6 ONS B3:3/3 MOV L13:6 L23:31 EOR
%   B3:7/6  CHUTE_OPT  "Stable chute optic output" %
%   B3:3/3  "one shot" %
%   L13:6  VIRT_TMR_BLOW2CHUTE  "count of time in ms for the blow to chute time" %
%   L23:31  BLOW2CHUTE_TIME %
% Rung: 4 %
SOR END EOR

LADDER 28 "FAULTS"
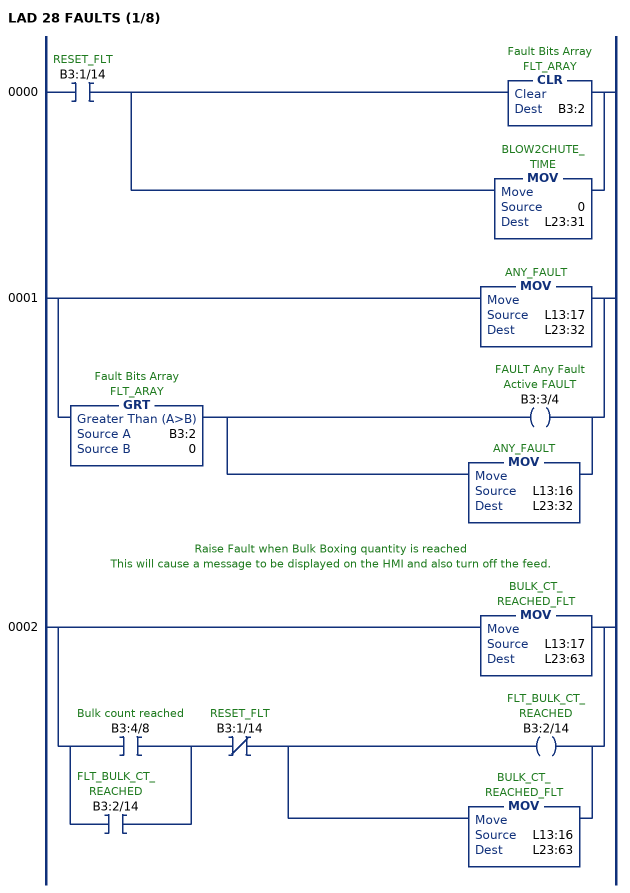
% Rung: 0 %
SOR XIC B3:1/14 BST CLR B3:2 NXB MOV 0 L23:31 BND EOR
%   B3:1/14  RESET_FLT %
%   B3:2  FLT_ARAY  "Fault Bits Array" %
%   L23:31  BLOW2CHUTE_TIME %
% Rung: 1 %
SOR BST MOV L13:17 L23:32 NXB GRT B3:2 0 BST OTE B3:3/4 NXB MOV L13:16 L23:32 BND BND EOR
%   L13:17  FALSE %
%   L23:32  ANY_FAULT %
%   B3:2  FLT_ARAY  "Fault Bits Array" %
%   B3:3/4  FAULT  "FAULT Any Fault Active" %
%   L13:16  TRUE  "ONE TIME ENABLE FOR THE TIMES WHEN WE FORGET TO RE-ENABLE AFTER SHIPMENT" %
% Rung: 2 %
% Raise Fault when Bulk Boxing quantity is reached
% 
% This will cause a message to be displayed on the HMI and also turn off the feed. %
SOR BST MOV L13:17 L23:63 NXB BST XIC B3:4/8 NXB XIC B3:2/14 BND XIO B3:1/14 BST OTE B3:2/14 NXB MOV L13:16 L23:63 BND BND EOR
%   L13:17  FALSE %
%   L23:63  BULK_CT_REACHED_FLT %
%   B3:4/8  "Bulk count reached" %
%   B3:2/14  FLT_BULK_CT_REACHED %
%   B3:1/14  RESET_FLT %
%   L13:16  TRUE  "ONE TIME ENABLE FOR THE TIMES WHEN WE FORGET TO RE-ENABLE AFTER SHIPMENT" %

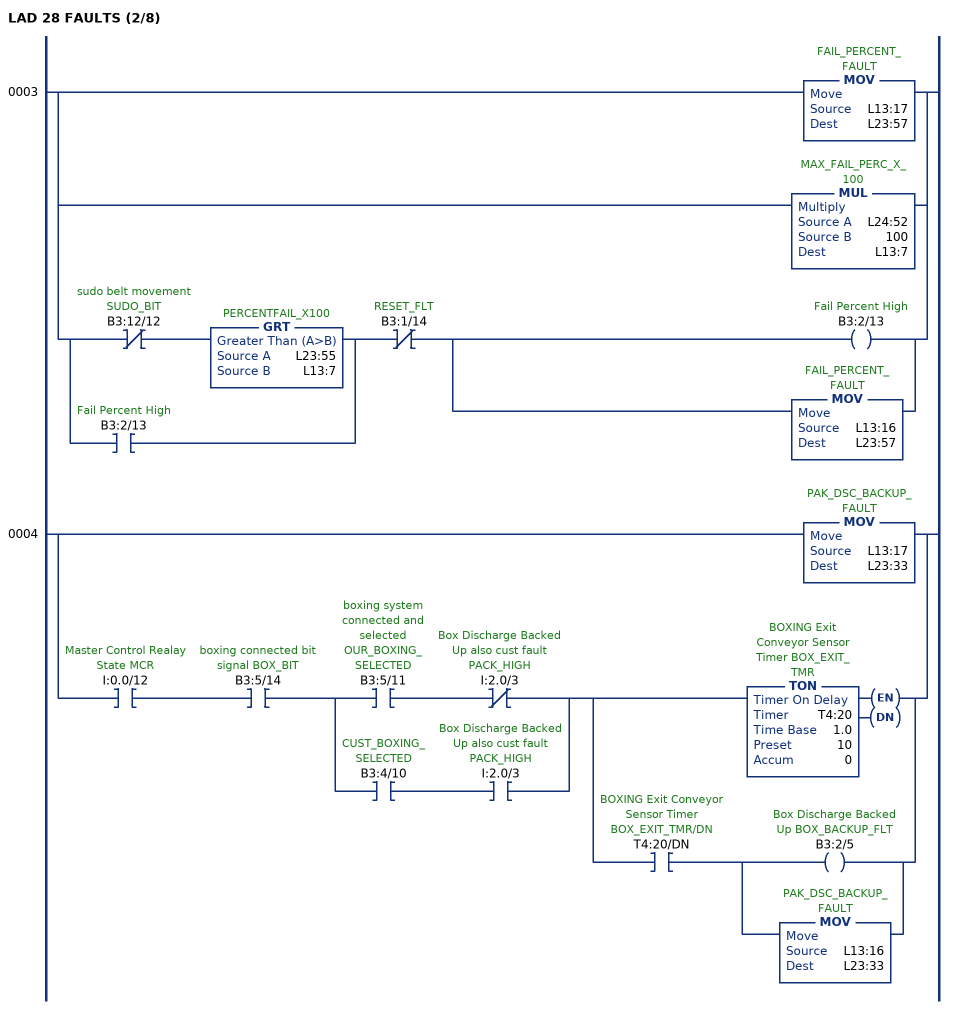
% Rung: 3 %
SOR BST MOV L13:17 L23:57 NXB MUL L24:52 100 L13:7 NXB BST XIO B3:12/12 GRT L23:55 L13:7 NXB XIC B3:2/13 BND XIO B3:1/14 BST OTE B3:2/13 NXB MOV L13:16 L23:57 BND BND EOR
%   L13:17  FALSE %
%   L23:57  FAIL_PERCENT_FAULT %
%   L24:52  MAX_FAIL_PERCENT %
%   L13:7  MAX_FAIL_PERC_X_100 %
%   B3:12/12  SUDO_BIT  "sudo belt movement" %
%   L23:55  PERCENTFAIL_X100 %
%   B3:2/13  "Fail Percent High" %
%   B3:1/14  RESET_FLT %
%   L13:16  TRUE  "ONE TIME ENABLE FOR THE TIMES WHEN WE FORGET TO RE-ENABLE AFTER SHIPMENT" %
% Rung: 4 %
SOR BST MOV L13:17 L23:33 NXB XIC I:0.0/12 XIC B3:5/14 BST XIC B3:5/11 XIO I:2.0/3 NXB XIC B3:4/10 XIC I:2.0/3 BND BST TON T4:20 1.0 10 0 NXB XIC T4:20/DN BST OTE B3:2/5 NXB MOV L13:16 L23:33 BND BND BND EOR
%   L13:17  FALSE %
%   L23:33  PAK_DSC_BACKUP_FAULT %
%   I:0.0/12  MCR  "Master Control Realay State" %
%   B3:5/14  BOX_BIT  "boxing connected bit signal" %
%   B3:5/11  OUR_BOXING_SELECTED  "boxing system connected and selected" %
%   I:2.0/3  PACK_HIGH  "Box Discharge Backed Up also cust fault" %
%   B3:4/10  CUST_BOXING_SELECTED %
%   T4:20  BOX_EXIT_TMR  "BOXING Exit Conveyor Sensor Timer" %
%   B3:2/5  BOX_BACKUP_FLT  "Box Discharge Backed Up" %
%   L13:16  TRUE  "ONE TIME ENABLE FOR THE TIMES WHEN WE FORGET TO RE-ENABLE AFTER SHIPMENT" %

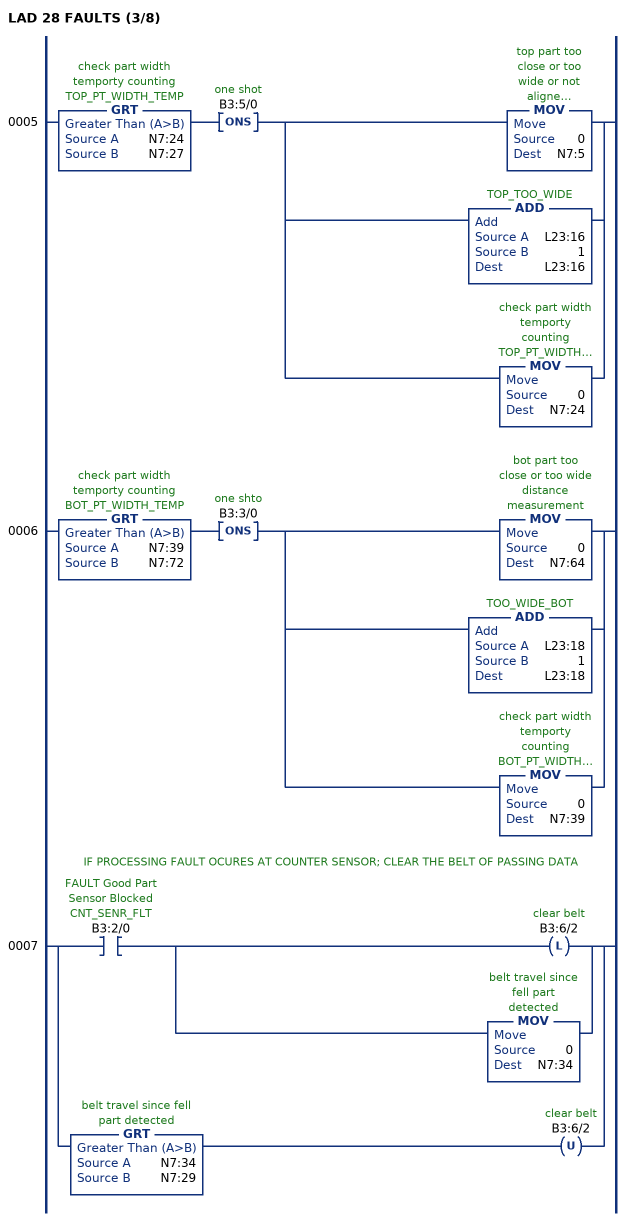
% Rung: 5 %
SOR GRT N7:24 N7:27 ONS B3:5/0 BST MOV 0 N7:5 NXB ADD L23:16 1 L23:16 NXB MOV 0 N7:24 BND EOR
%   N7:24  TOP_PT_WIDTH_TEMP  "check part width temporty counting" %
%   N7:27  "max part width top optic" %
%   B3:5/0  "one shot" %
%   N7:5  "top part too close or too wide or not aligned distance measurement" %
%   L23:16  TOP_TOO_WIDE %
% Rung: 6 %
SOR GRT N7:39 N7:72 ONS B3:3/0 BST MOV 0 N7:64 NXB ADD L23:18 1 L23:18 NXB MOV 0 N7:39 BND EOR
%   N7:39  BOT_PT_WIDTH_TEMP  "check part width temporty counting" %
%   N7:72  "max part width bottom optic" %
%   B3:3/0  "one shto" %
%   N7:64  "bot part too close or too wide distance measurement" %
%   L23:18  TOO_WIDE_BOT %
% Rung: 7 %
% IF PROCESSING FAULT OCURES AT COUNTER SENSOR; CLEAR THE BELT OF PASSING DATA %
SOR BST XIC B3:2/0 BST OTL B3:6/2 NXB MOV 0 N7:34 BND NXB GRT N7:34 N7:29 OTU B3:6/2 BND EOR
%   B3:2/0  CNT_SENR_FLT  "FAULT Good Part Sensor Blocked" %
%   B3:6/2  "clear belt" %
%   N7:34  "belt travel since fell part detected" %
%   N7:29  "belt travel to wipe parts off of belt when fell part detected" %

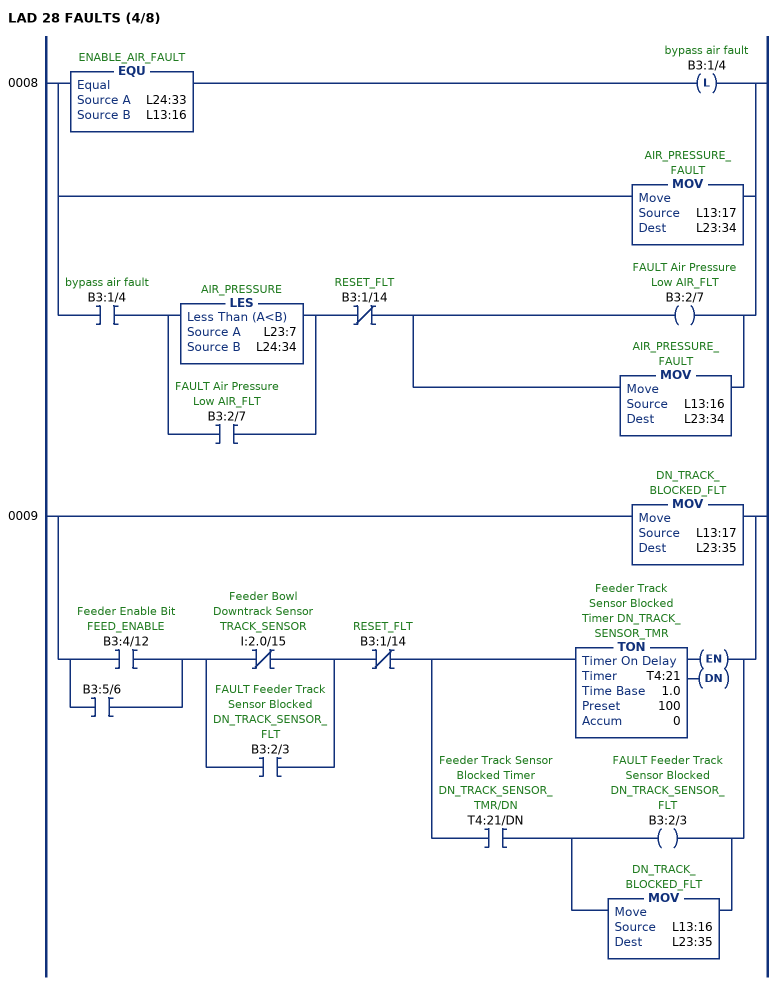
% Rung: 8 %
SOR BST EQU L24:33 L13:16 OTL B3:1/4 NXB MOV L13:17 L23:34 NXB XIC B3:1/4 BST LES L23:7 L24:34 NXB XIC B3:2/7 BND XIO B3:1/14 BST OTE B3:2/7 NXB MOV L13:16 L23:34 BND BND EOR
%   L24:33  ENABLE_AIR_FAULT %
%   L13:16  TRUE  "ONE TIME ENABLE FOR THE TIMES WHEN WE FORGET TO RE-ENABLE AFTER SHIPMENT" %
%   B3:1/4  "bypass air fault" %
%   L13:17  FALSE %
%   L23:34  AIR_PRESSURE_FAULT %
%   L23:7  AIR_PRESSURE %
%   L24:34  MIN_AIR_PRESSURE %
%   B3:2/7  AIR_FLT  "FAULT Air Pressure Low" %
%   B3:1/14  RESET_FLT %
% Rung: 9 %
SOR BST MOV L13:17 L23:35 NXB BST XIC B3:4/12 NXB XIC B3:5/6 BND BST XIO I:2.0/15 NXB XIC B3:2/3 BND XIO B3:1/14 BST TON T4:21 1.0 100 0 NXB XIC T4:21/DN BST OTE B3:2/3 NXB MOV L13:16 L23:35 BND BND BND EOR
%   L13:17  FALSE %
%   L23:35  DN_TRACK_BLOCKED_FLT %
%   B3:4/12  FEED_ENABLE  "Feeder Enable Bit" %
%   I:2.0/15  TRACK_SENSOR  "Feeder Bowl Downtrack Sensor" %
%   B3:2/3  DN_TRACK_SENSOR_FLT  "FAULT Feeder Track Sensor Blocked" %
%   B3:1/14  RESET_FLT %
%   T4:21  DN_TRACK_SENSOR_TMR  "Feeder Track Sensor Blocked Timer" %
%   L13:16  TRUE  "ONE TIME ENABLE FOR THE TIMES WHEN WE FORGET TO RE-ENABLE AFTER SHIPMENT" %

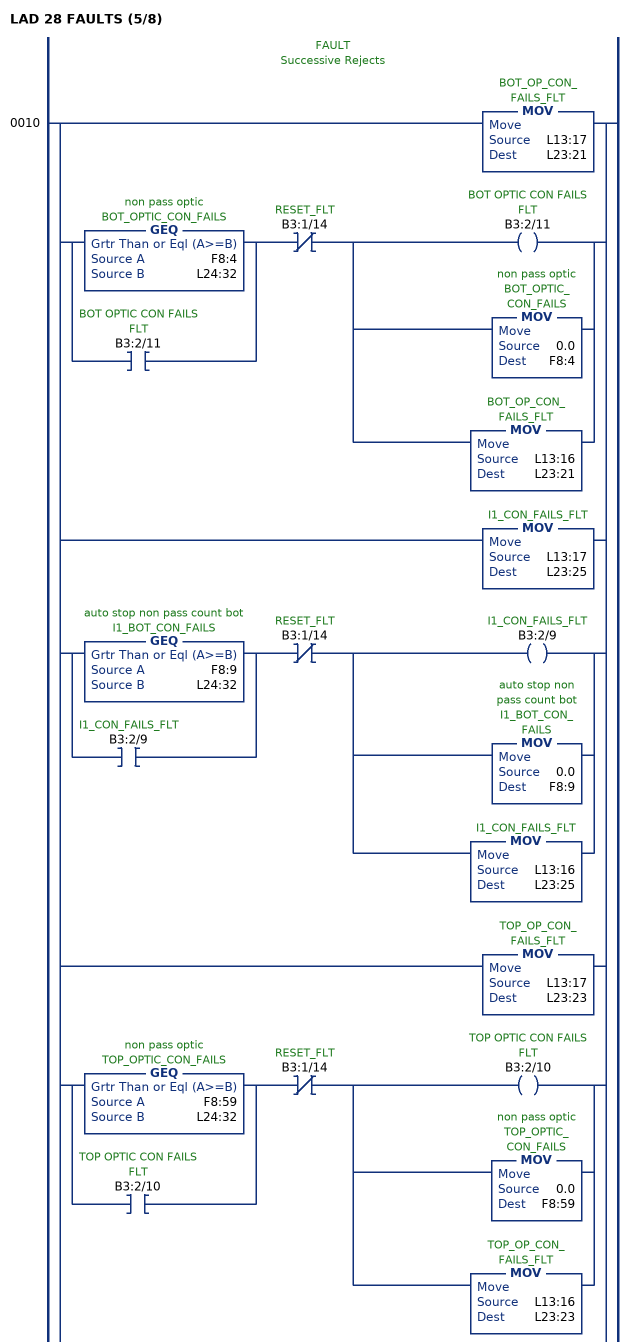

